(* IEC 61131-3 sources: ATCMcontrol_Engineering/src/COM/softing/fc/CL/Libs/ATCM_IEC1131_3/table_35, 2 files *)

(* ---- f_trig.st ---- *)
(*[[
    UserURL= "ATCMFile:F_TRIG.htm"
]]*)
FUNCTION_BLOCK F_TRIG
VAR_INPUT
	CLK: BOOL;
END_VAR
VAR_OUTPUT
	Q: BOOL;
END_VAR
VAR
	M: BOOL := TRUE;
END_VAR

Q := NOT CLK AND NOT M;
M := NOT CLK;

END_FUNCTION_BLOCK

(* ---- r_trig.st ---- *)
(*[[
    UserURL= "ATCMFile:R_TRIG.htm"
]]*)
FUNCTION_BLOCK R_TRIG
VAR_INPUT
	CLK: BOOL;
END_VAR
VAR_OUTPUT
	Q: BOOL;
END_VAR
VAR
	M: BOOL := FALSE;
END_VAR

Q := CLK AND NOT M;
M := CLK;

END_FUNCTION_BLOCK
